// SIMATIC S7-200 project (STEP 7-Micro/WIN), CPU 221 REL 01.10

ORGANIZATION_BLOCK 主程序:OB1
TITLE=程序注释
BEGIN
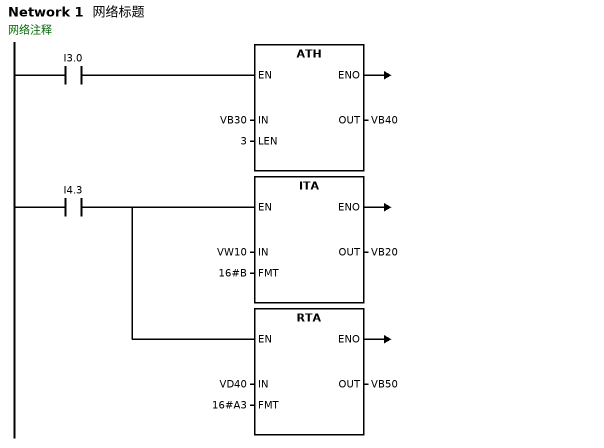
Network 1 // 网络标题
// 网络注释
// (network saved uncompiled; LAD cells follow)
// row 0: c0 -| |- I3.0  c1 --  c2 [ATH EN:=power@row0, IN:=VB30, LEN:=3, ENO=>power, OUT=>VB40]  c3 ->
// row 1: c2 [box]
// row 2: c0 -| |- I4.3 v  c1 --  c2 [ITA EN:=power@row2, IN:=VW10, FMT:=16#B, ENO=>power, OUT=>VB20]  c3 ->
// row 3: c0 ^v  c2 [box]
// row 4: c0 ^  c1 --  c2 [RTA EN:=power@row4, IN:=VD40, FMT:=16#A3, ENO=>power, OUT=>VB50]  c3 ->
// row 5: c2 [box]
END_ORGANIZATION_BLOCK
